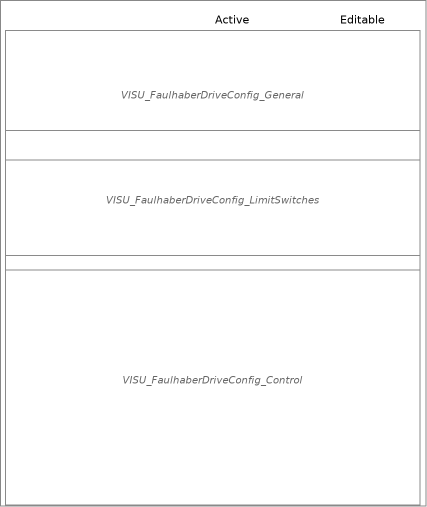
VISUALIZATION VISU_FaulhaberDriveConfig  // 427x507
VAR_IN_OUT
	active : FaulhaberDriveConfig;
	editable : FaulhaberDriveConfig;
END_VAR
    Frame (5,30 415x130)
        shows VISU_FaulhaberDriveConfig_General(active := active, editable := editable)
        shows VISU_FaulhaberDriveConfig_Control(active := active, editable := editable)
        shows VISU_FaulhaberDriveConfig_LimitSwitches(active := active, editable := editable)
    Frame (5,255 415x250)
        shows VISU_FaulhaberDriveConfig_Control(active := active, editable := editable)
        shows VISU_FaulhaberDriveConfig_LimitSwitches(active := active, editable := editable)
        p1986482694: active
        p3357690139: editable
    Frame (5,130 415x140)
        shows VISU_FaulhaberDriveConfig_LimitSwitches(active := active, editable := editable)
        shows VISU_FaulhaberDriveConfig_Control(active := active, editable := editable)
        p1340763843: active
        p1371549466: editable
    Label (170,10 125x20), "Active"
    Label (300,10 125x20), "Editable"
END_VISUALIZATION

(* stored: Version 1.1.0.1, ProductVersion 3.1.4019.2
   Visu VISU_FaulhaberDriveConfig: Id {2fb5b718-fc6c-4f7e-870e-bb3b13b7604c} *)
